{attribute 'GeneratedUsingTerminal: EL7211-0010-0032'}
{attribute addProperty BoxType "EL7211-0010-0032"}
{attribute addProperty Id "StatuswordAT %I*UINT2"}
{attribute addProperty CRC "2604072444"}
{attribute addProperty Size "2"}
TYPE DRV_Statusword_9B36FDFC EXTENDS TcoIo.InputBase_8311D824 :
STRUCT
	{attribute addProperty Name "Statusword"}
	Statusword AT %I* : UINT;
END_STRUCT
END_TYPE

(* stored: Version 1.2.0.0, ProductVersion 3.1.4024.11
   DUT DRV_Statusword_9B36FDFC: Id {b3e04b3f-fb90-01fe-0031-0101a270a4ea} *)
